{attribute 'GeneratedUsingTerminal: EL7211-0010-0032'}
{attribute addProperty BoxType "EL7211-0010-0032"}
{attribute addProperty Id "PositionAT %I*UDINT4"}
{attribute addProperty CRC "1067488493"}
{attribute addProperty Size "4"}
TYPE FB_Position_3FA094ED EXTENDS TcoIo.InputBase_8311D824 :
STRUCT
	{attribute addProperty Name "Position"}
	Position AT %I* : UDINT;
END_STRUCT
END_TYPE

(* stored: Version 1.2.0.0, ProductVersion 3.1.4024.11
   DUT FB_Position_3FA094ED: Id {a5778ac4-a4cf-0149-1e57-150a8c6c100e} *)
